FUNCTION_BLOCK RunClamper EXTENDS RunUnitSlave
VAR_INPUT
	scaraAck at%Q* : bool; //SCARA acknowledge feed-in part
END_VAR
VAR_OUTPUT
END_VAR
VAR
	//devices
	horizon : POINTER TO RunCylinder;
	clamper : POINTER TO RunCylinder;
	//
	configSnap : BOOL; //set true for instance of Snap
	
END_VAR
VAR CONSTANT
	bScaraReady : INT := 1;
END_VAR

SUPER^();

//Link to :
// 1. Indexer - working signal
// 2. Bridge - working signal dispatch  to SCARA

CASE outputState OF
	//---------------------------
	//	Initialization : hold and push
	//---------------------------	
	eSpecialStates.INITIAL_BEGIN:
		bSerialTransition := clamper^.Execute(eCylinderCommands.COMMAND_A);
	eSpecialStates.INITIAL_STATE_1:
		bSerialTransition := horizon^.Execute(eCylinderCommands.COMMAND_A);
	eSpecialStates.INITIAL_STATE_2:
		bSerialTransition := clamper^.Execute(eCylinderCommands.COMMAND_B); //hold
	eSpecialStates.INITIAL_STATE_3:
		bSerialTransition := horizon^.Execute(eCylinderCommands.COMMAND_B); //push
	eSpecialStates.INITIAL_STATE_5:
		bSerialTransition := clamper^.Execute(eCylinderCommands.COMMAND_A);	//release 
	eSpecialStates.INITIAL_STATE_6:
		bSerialTransition := horizon^.Execute(eCylinderCommands.COMMAND_A);	//back 
		IF bSerialTransition THEN
			NextState := eSpecialStates.INITIAL_END;
		END_IF
	//----------------------------
	//	Working
	//----------------------------
	eSpecialStates.SLAVE_ENTER_PROCEDURE:
		IF SlotBase^.Valid THEN
			bSerialTransition := TRUE;
		ELSE
			NextState := 16#205; //bypass
		END_IF
	16#201:
		//Indexer in position , horizonin
		bSerialTransition := horizon^.Execute(eCylinderCommands.COMMAND_B);
	16#202:
		bSerialTransition := clamper^.Execute(eCylinderCommands.COMMAND_B);
	16#203:
		transitionByte.0 := horizon^.Execute(eCylinderCommands.COMMAND_A);
		//----------------------
		//	Snapping fit special 
		//----------------------
		IF configSnap THEN
			transitionByte.1 := clamper^.Execute(eCylinderCommands.COMMAND_A);
		ELSE
			transitionByte.1 := TRUE;	
		END_IF
		
		IF transitionByte = 16#3 THEN
			slaveWorkingSignal[bScaraReady]:= TRUE; //trigger SCARA agent
			bSerialTransition := TRUE;
		END_IF
	16#204:
		//Wait SCARA 
		bSerialTransition := NOT slaveWorkingSignal[bScaraReady];
	16#205:
		//send part back to indexer
		bSerialTransition := horizon^.Execute(eCylinderCommands.COMMAND_B);
	16#206:
		//release part 
		bSerialTransition := clamper^.Execute(eCylinderCommands.COMMAND_A); //release
	16#207:
		//empty clamper extract
		IF horizon^.Execute(eCylinderCommands.COMMAND_A) THEN
			NextState := eSpecialStates.SLAVE_WORK_DONE;
		END_IF
END_CASE

METHOD FB_init : BOOL
VAR_INPUT
	bInitRetains : BOOL; // if TRUE, the retain variables are initialized (warm start / cold start)
	bInCopyCode : BOOL;  // if TRUE, the instance afterwards gets moved into the copy code (online change)
	
	argParent : POINTER TO RunUnitGeneric;
	argSlotBase : POINTER TO RunMaterial;
	argSlotLast : POINTER TO RunMaterial;
	
	argWorkingSignal : POINTER TO BOOL;
	
	argHorizon : POINTER TO RunCylinder;
	argClamper : POINTER TO RunCylinder;
	argConfigSnap : BOOL;
END_VAR
//initialize 
Parent := argParent;
SlotBase := argSlotBase;
SlotLast := argSlotLast;
//
IF bInitRetains THEN
	NextState := eSpecialStates.INITIAL_BEGIN;
END_IF

workingSignal := argWorkingSignal; //link

//device link
horizon := argHorizon;
clamper := argClamper;
configSnap := argConfigSnap;
END_METHOD

END_FUNCTION_BLOCK

(* stored: Version 1.1.0.1, ProductVersion 3.1.4024.0
   POU RunClamper: Id {4cfbb8e7-dd19-45d2-8e96-6129406da078}, SpecialFunc None
   Method FB_init: Id {37c62737-651a-4f40-81e3-f79b76fcc99a} *)
